FUNCTION TryConvert_ULINT_TO_TOD : BOOL
VAR_INPUT
	in : ULINT;
	out : REFERENCE TO TOD;
END_VAR

IF in > DatatypeLimits.MAX_VALUE_OF_ULINT_WHICH_CAN_BE_HELD_IN_A_TOD THEN
	RETURN;
END_IF

out := ULINT_TO_TOD(in);
TryConvert_ULINT_TO_TOD := TRUE;

END_FUNCTION

(* stored: Version 1.1.0.1, ProductVersion 3.1.4024.12
   POU TryConvert_ULINT_TO_TOD: Id {9994dee5-ff46-4b9d-9e19-db998ad13f1a}, SpecialFunc None *)
